// TIA Portal project "2_Box_Sorting_Height" (V19)

(* hardware
DEVICE "S7-1500/ET200MP station_1"  S7-1500 station
   slot 0: "Rail_0"  Rack  6ES7 590-1***0-0AA0
   slot 1: "PLC_1"  CPU 1513-1 PN  6ES7 513-1AL02-0AB0  V2.9
      slot 3: "CPU display_1"  6ES7591-1AA00-0AA0
      slot 32768: "PROFINET interface_1"  X1
         slot 32769: "Port_1"  X1 P1
         slot 32770: "Port_2"  X1 P2
      slot 34817: "Virtual CP interface port_1"  Virtual CP interface port  Virtual CP interface port
*)

// ===== PLC "PLC_1"  CPU 1513-1 PN =====

VAR_GLOBAL   // PLC tag table "Default tag table"
   "SR Memory" AT %M0.0 : Bool;
   "NGE_Height Sensor" AT %M0.1 : Bool;
   "NGE_Large Box Counting Sensor" AT %M0.2 : Bool;
   "NGE_Small Box Counting Sensor(1)" AT %M0.3 : Bool;
   "Timer O/P to RS from ON position" AT %M0.4 : Bool;
   "M0.4 Buffer" AT %M0.5 : Bool;
   "Push Front" AT %I0.5 : Bool;
   "Timer O/P to RS from OFF position" AT %M0.6 : Bool;
   "M0.6 Buffer" AT %M0.7 : Bool;
   "M0.6 buffer with NGE" AT %M1.0 : Bool;
END_VAR

VAR_GLOBAL   // PLC tag table "Tag table from XML_4"
   "Start" AT %I0.0 : Bool;
   "Stop" AT %I0.1 : Bool;
   "Height Sensor" AT %I0.2 : Bool;
   "Large Box Sensor" AT %I0.3 : Bool;
   "Small Box Sensor" AT %I0.4 : Bool;
   "Reset" AT %I0.6 : Bool;
   "Conveyor Belt" AT %Q0.0 : Bool;
   "Emitter" AT %Q0.1 : Bool;
   "Pusher" AT %Q0.2 : Bool;
   "Start (Light)" AT %Q0.3 : Bool;
   "Stop  (Light)" AT %Q0.4 : Bool;
   "Reset (Light)" AT %Q0.5 : Bool;
   "Large Box Count" AT %QD30 : DInt;
   "Small Box Count" AT %QD34 : DInt;
END_VAR

// folder: System blocks/Program resources

DATA_BLOCK "IEC_Counter_0_DB"   // DB1
{ S7_Optimized_Access := 'TRUE' }
AUTHOR : SIMATIC
FAMILY : IEC
NAME : DCNTR
VERSION : 1.2
// stored: InstanceOfName IEC_DCOUNTER
"IEC_DCOUNTER"
BEGIN
END_DATA_BLOCK

DATA_BLOCK "IEC_Counter_0_DB_1"   // DB2
{ S7_Optimized_Access := 'TRUE' }
AUTHOR : SIMATIC
FAMILY : IEC
NAME : DCNTR
VERSION : 1.2
// stored: InstanceOfName IEC_DCOUNTER
"IEC_DCOUNTER"
BEGIN
END_DATA_BLOCK

DATA_BLOCK "IEC_Timer_0_DB"   // DB3
{ S7_Optimized_Access := 'TRUE' }
AUTHOR : Simatic
FAMILY : IEC
NAME : IEC_TMR
VERSION : 1.0
// stored: InstanceOfName IEC_TIMER
"IEC_TIMER"
BEGIN
END_DATA_BLOCK

DATA_BLOCK "IEC_Timer_0_DB_1"   // DB4
{ S7_Optimized_Access := 'TRUE' }
AUTHOR : Simatic
FAMILY : IEC
NAME : IEC_TMR
VERSION : 1.0
// stored: InstanceOfName IEC_TIMER
"IEC_TIMER"
BEGIN
END_DATA_BLOCK

// folder: (top level)

ORGANIZATION_BLOCK "Main"   // OB1, LAD, ProgramCycle
TITLE = "Main Program Sweep (Cycle)"
{ S7_Optimized_Access := 'TRUE' }
VERSION : 0.1
   VAR_INPUT
      Initial_Call : Bool;   // Initial call of this OB
      Remanence : Bool;   // =True, if remanent data are available
   END_VAR
   VAR_TEMP   // added for the SCL form of the ladder/FBD networks
      _w1 : Bool;
      _w2 : Bool;
      _w3 : Bool;
   END_VAR
BEGIN

REGION Network 1
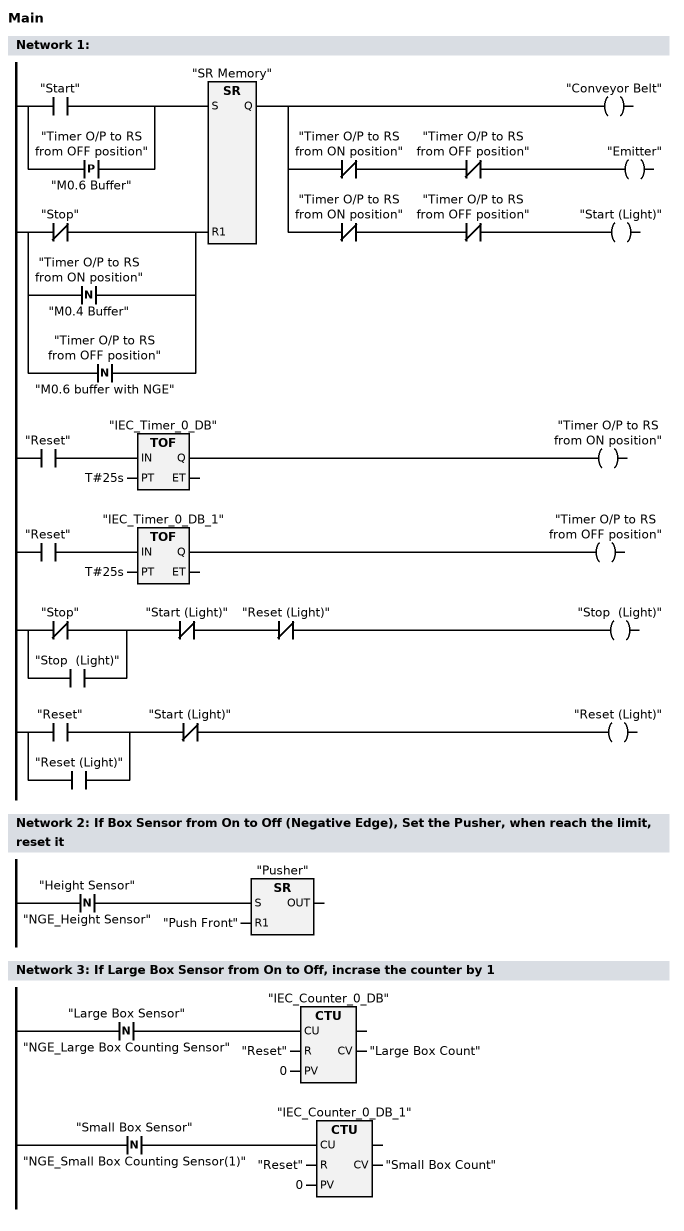
   #_w1 := "Timer O/P to RS from OFF position" AND NOT "M0.6 Buffer";   // rising edge of "Timer O/P to RS from OFF position"
   "M0.6 Buffer" := "Timer O/P to RS from OFF position";
   #_w2 := NOT "Timer O/P to RS from ON position" AND "M0.4 Buffer";   // falling edge of "Timer O/P to RS from ON position"
   "M0.4 Buffer" := "Timer O/P to RS from ON position";
   #_w3 := NOT "Timer O/P to RS from OFF position" AND "M0.6 buffer with NGE";   // falling edge of "Timer O/P to RS from OFF position"
   "M0.6 buffer with NGE" := "Timer O/P to RS from OFF position";
   IF "Start" OR #_w1 THEN
       "SR Memory" := TRUE;   // SR flip-flop
   END_IF;
   IF NOT "Stop" OR #_w2 OR #_w3 THEN "SR Memory" := FALSE; END_IF;
   "Conveyor Belt" := "SR Memory";
   "Emitter" := "SR Memory" AND NOT "Timer O/P to RS from ON position" AND NOT "Timer O/P to RS from OFF position";
   "Start (Light)" := "SR Memory" AND NOT "Timer O/P to RS from ON position" AND NOT "Timer O/P to RS from OFF position";
   "IEC_Timer_0_DB".TOF(IN := "Reset", PT := T#25s);
   "Timer O/P to RS from ON position" := "IEC_Timer_0_DB".Q;
   "IEC_Timer_0_DB_1".TOF(IN := "Reset", PT := T#25s);
   "Timer O/P to RS from OFF position" := "IEC_Timer_0_DB_1".Q;
   "Stop  (Light)" := (NOT "Stop" OR "Stop  (Light)") AND NOT "Start (Light)" AND NOT "Reset (Light)";
   "Reset (Light)" := ("Reset" OR "Reset (Light)") AND NOT "Start (Light)";
END_REGION

REGION Network 2: If Box Sensor from On to Off (Negative Edge), Set the Pusher, when reach the limit, reset it
   RUNG wire#powerrail
      N_Contact(operand := "Height Sensor", bit := "NGE_Height Sensor")
      S_SR(operand := "Pusher", r1 := "Push Front")
   END_RUNG
   // the same network as SCL:
   #_w1 := NOT "Height Sensor" AND "NGE_Height Sensor";   // falling edge of "Height Sensor"
   "NGE_Height Sensor" := "Height Sensor";
   IF #_w1 THEN
       "Pusher" := TRUE;   // SR flip-flop
   END_IF;
   IF "Push Front" THEN "Pusher" := FALSE; END_IF;
END_REGION

REGION Network 3: If Large Box Sensor from On to Off, incrase the counter by 1
   #_w1 := NOT "Large Box Sensor" AND "NGE_Large Box Counting Sensor";   // falling edge of "Large Box Sensor"
   "NGE_Large Box Counting Sensor" := "Large Box Sensor";
   "IEC_Counter_0_DB".CTU(CU := #_w1, R := "Reset", PV := 0, CV => "Large Box Count");
   #_w2 := NOT "Small Box Sensor" AND "NGE_Small Box Counting Sensor(1)";   // falling edge of "Small Box Sensor"
   "NGE_Small Box Counting Sensor(1)" := "Small Box Sensor";
   "IEC_Counter_0_DB_1".CTU(CU := #_w2, R := "Reset", PV := 0, CV => "Small Box Count");
END_REGION
END_ORGANIZATION_BLOCK